// TIA Portal V17 export
// export: Created 2025-08-05T09:36:01.9783417Z, ExportSetting WithDefaults, DisplayName Totally Integrated Automation Portal, DisplayVersion V17, DisplayName TIA Portal Openness, DisplayVersion V17, DisplayName TIA Portal Version Control Interface, DisplayVersion V17, DisplayName SINAMICS Startdrive Advanced, DisplayVersion V17, DisplayName SINAMICS Startdrive G130, G150, S120, S150, SINAMICS MV, S210, DisplayVersion V17, DisplayName SINAMICS Startdrive G110M, G120, G120C, G120D, G120P, G115D, DisplayVersion V17, DisplayName STEP 7 Professional, DisplayVersion V17, DisplayName STEP 7 Safety, DisplayVersion V17, DisplayName WinCC Advanced, DisplayVersion V17
TYPE "YLS_Outputs"
// stored: IsFailsafeCompliant false
   STRUCT
      Laser_Request : Bool;   // Laser_Request
      Laser_On : Bool;   // Laser_On
      Reset_Errors : Bool;   // Reset_Errors
      Guide_Laser_On : Bool;   // Guide_Laser_On
      Program_Start : Bool;   // Program_Start
      Program_Stop : Bool;   // Program_Stop
      Reserved : Bool;   // Reserved
      Analogue_Control_On : Bool;   // Analogue_Control_On
      Control_by_LaserNet : Bool;   // Control_by_LaserNet
      Set_Rise_Time : Bool;   // Set_Rise_Time
      Set_Fall_Time : Bool;   // Set_Fall_Time
      Synchronization_Input : Bool;   // Synchronization_Input
      Reserved_1 : Bool;   // Reserved_1
      Piercing_Mode : Bool;   // Piercing_Mode
      Single_Module_Mode : Bool;   // Single_Module_Mode
      External_Error : Bool;   // External_Error
      Power : Int;   // Power
      Optical_Channel : Byte;   // Optical_Channel
      Program_Number : Byte;   // Program_Number
      Ramping_Time : Int;   // Ramping_Time
      Laser_Number : Byte;   // Laser_Number
      Reserved_2 : Byte;   // Reserved_2
      Modules_Selection : Int;   // Modules_Selection
      Core_Modules_Power_Setpoint : Int;   // Core_Modules_Power_Setpoint
      Ring_Modules_Power_Setpoint : Int;   // Ring_Modules_Power_Setpoint
   END_STRUCT;
END_TYPE
